{attribute 'qualified_only'}
VAR_GLOBAL
	stBoxParam : ST_BoxParam;
	
END_VAR

(* stored: Version 1.1.0.1, ProductVersion 3.1.4024.12
   GVL Input: Id {11a78f26-7726-48b1-9eef-c95b38186742} *)
